INTERFACE I_StructuredDatatypeAddedEvent EXTENDS I_Event

PROPERTY PUBLIC Target : I_StructuredDatatype
GET
END_GET
END_PROPERTY

END_INTERFACE

(* stored: Version 1.1.0.1, ProductVersion 3.1.4024.12
   Itf I_StructuredDatatypeAddedEvent: Id {fbd431c4-bb56-0e10-158f-d14d28592616}
   Property Target: Id {df1db57e-89b6-05de-1584-5c2695ea576a}
   Get Get: Id {1817503e-1d2d-0548-1373-c049d783c4d4} *)
